
// ===== library: MasterCopy "Turbina" =====

FUNCTION_BLOCK "Turbina"   // FB1, LAD
{ S7_Optimized_Access := 'TRUE' }
VERSION : 0.1
   VAR_INPUT
      MotorAuxiliar : Bool;
      JuntaNeum : Bool;
      Frenos : Bool;
      Quemador_A : Bool;   // Entrada digital - Sensor Quemador A
      Quemador_B : Bool;   // Entrada digital - Sensor Quemador B
      Reset : Bool := False;
      ModoControl : Bool;   // Modo de control = 0=Manual 1=Auto
      SPManual : Int;   // Consigna manual
      SPAuto : Int;   // Consigna Automatica
   END_VAR
   VAR_OUTPUT
      SalidaVel : Int;
      SalidaPres : Int;
   END_VAR
   VAR_IN_OUT
      DB_Lazo : PID_Compact;
   END_VAR
   VAR
      Comando : Real;
      VelReal : Real;
      ValvReal : Real;
      ModeloPlanta : "ModeloPlanta";
      SP_ManualReal : Real;
      Valvula : Int;
      SP_AutoReal : Real;
   END_VAR
   VAR_TEMP
      KFrenos : Real;
      KMotor : Real;
      state : Int;
      error : Bool;
   END_VAR
   VAR_TEMP   // added for the SCL form of the ladder/FBD networks
      _w1 : Bool;
   END_VAR
BEGIN

REGION Network 1
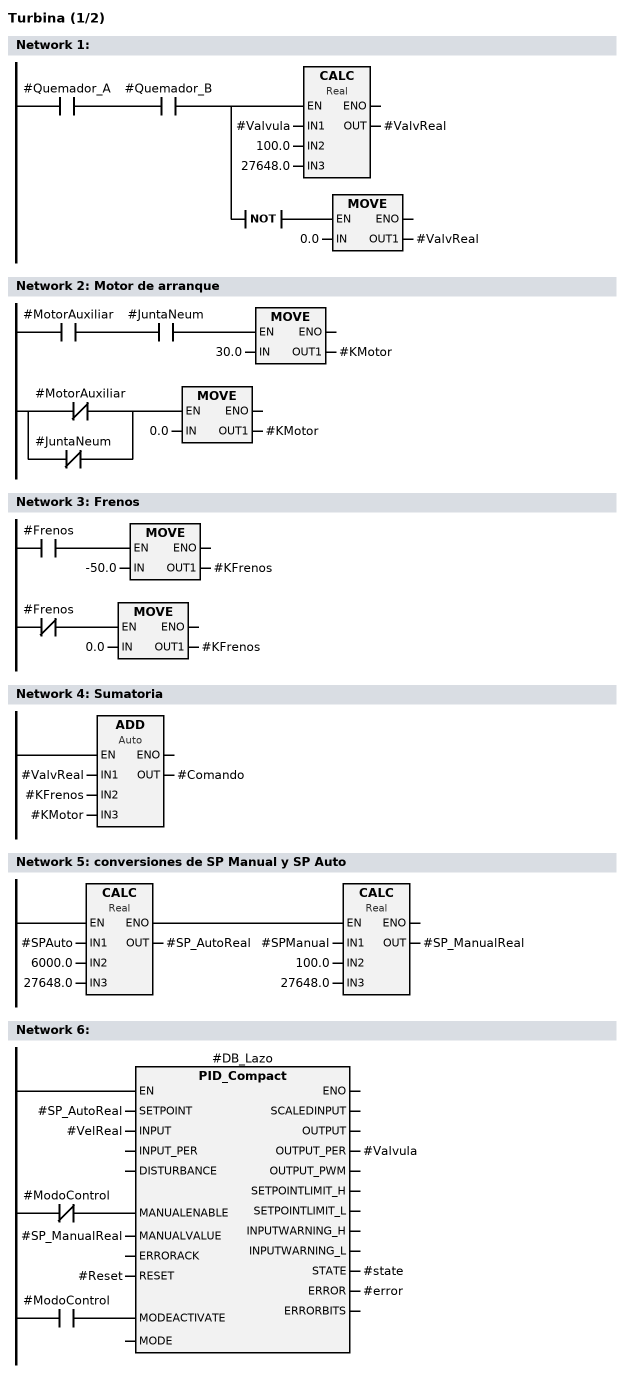
   #_w1 := #Quemador_A AND #Quemador_B;
   IF #_w1 THEN CALC(in1 := #Valvula, in2 := 100.0, in3 := 27648.0, out => #ValvReal); END_IF;
   IF NOT #_w1 THEN #ValvReal := 0.0; END_IF;
END_REGION

REGION Network 2: Motor de arranque
   RUNG wire#powerrail
      Contact( #MotorAuxiliar )
      Contact( #JuntaNeum )
      Move(in := 30.0, out1 => #KMotor)
   END_RUNG
   RUNG wire#powerrail
      I_Contact( #MotorAuxiliar )
      wire#w1
      Move(in := 0.0, out1 => #KMotor)
   END_RUNG
   RUNG wire#powerrail
      I_Contact( #JuntaNeum )
   END_RUNG wire#w1
   // the same network as SCL:
   IF #MotorAuxiliar AND #JuntaNeum THEN #KMotor := 30.0; END_IF;
   IF NOT #MotorAuxiliar OR NOT #JuntaNeum THEN #KMotor := 0.0; END_IF;
END_REGION

REGION Network 3: Frenos
   RUNG wire#powerrail
      Contact( #Frenos )
      Move(in := -50.0, out1 => #KFrenos)
   END_RUNG
   RUNG wire#powerrail
      I_Contact( #Frenos )
      Move(in := 0.0, out1 => #KFrenos)
   END_RUNG
   // the same network as SCL:
   IF #Frenos THEN #KFrenos := -50.0; END_IF;
   IF NOT #Frenos THEN #KFrenos := 0.0; END_IF;
END_REGION

REGION Network 4: Sumatoria
   RUNG wire#powerrail
      Add(in1 := #ValvReal, in2 := #KFrenos, in3 := #KMotor, out => #Comando)
   END_RUNG
   // the same network as SCL:
   #Comando := #ValvReal + #KFrenos + #KMotor;
END_REGION

REGION Network 5: conversiones de SP Manual y SP Auto
   CALC(in1 := #SPAuto, in2 := 6000.0, in3 := 27648.0, out => #SP_AutoReal);
   CALC(in1 := #SPManual, in2 := 100.0, in3 := 27648.0, out => #SP_ManualReal);
END_REGION

REGION Network 6
   #DB_Lazo(Setpoint := #SP_AutoReal,   // PID_Compact
            Input := #VelReal,
            ManualEnable := NOT #ModoControl,
            ManualValue := #SP_ManualReal,
            Reset := #Reset,
            ModeActivate := #ModoControl,
            Output_PER => #Valvula,
            State => #state,
            Error => #error);
END_REGION

REGION Network 7
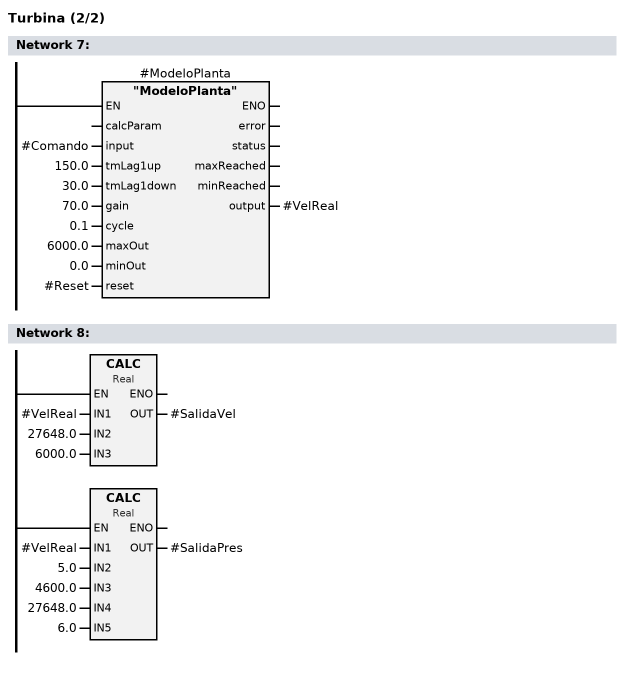
   RUNG wire#powerrail
      #ModeloPlanta(calcParam :=, input := #Comando, tmLag1up := 150.0, tmLag1down := 30.0, gain := 70.0, cycle := 0.1, maxOut := 6000.0, minOut := 0.0, reset := #Reset, error =>, status =>, maxReached =>, minReached =>, output => #VelReal)
   END_RUNG
   // the same network as SCL:
   #ModeloPlanta(input := #Comando,   // "ModeloPlanta"
                 tmLag1up := 150.0,
                 tmLag1down := 30.0,
                 gain := 70.0,
                 cycle := 0.1,
                 maxOut := 6000.0,
                 minOut := 0.0,
                 reset := #Reset,
                 output => #VelReal);
END_REGION

REGION Network 8
   CALC(in1 := #VelReal, in2 := 27648.0, in3 := 6000.0, out => #SalidaVel);
   CALC(in1 := #VelReal, in2 := 5.0, in3 := 4600.0, in4 := 27648.0, in5 := 6.0, out => #SalidaPres);
END_REGION
END_FUNCTION_BLOCK

// ===== library: MasterCopy "ModeloPlanta" =====

FUNCTION_BLOCK "ModeloPlanta"   // FB51, SCL
{ S7_Optimized_Access := 'TRUE' }
VERSION : 2.01
   VAR_INPUT
      calcParam : Bool;   // recalculate with new parameters
      input : Real;   // input signal
      tmLag1up : Real := 1.0;   // time constant T1 [sec] rising input
      tmLag1down : Real := 10.0;   // time constant T1 [sec] falling input
      gain : Real := 1.0;   // gain factor
      cycle : Real := 0.1;   // cyclic time [sec]
      maxOut : Real := 100.0;   // max. output limit
      minOut : Real;   // min. output limit
      reset : Bool;   // resets all relevant parameters to ‘0’ including the output
   END_VAR
   VAR_OUTPUT
      error : Bool;   // error (#tmLag1 <= 0 or #tmLag2 <= 0)
      status : Word;   // status (if #error = TRUE then status = 16#8001)
      maxReached : Bool;   // output has reached max. limit
      minReached : Bool;   // output has reached min. limit
      output : Real;   // output signal (if #error = FALSE)
   END_VAR
   VAR
      statRxn1 : Real;   // delayed input signal (n-1)
      statRyn1 : Real;   // delayed output signal (n-1)
      statRf1up : Real;   // Z-parameter 1 (rising xn)
      statRe1up : Real;   // Z-parameter 2 (rising xn)
      statRf1dn : Real;   // Z-parameter 1 (falling xn)
      statRe1dn : Real;   // Z-parameter 2 (falling xn)
      statRf1 : Real;   // active Z-parameter 1
      statRe1 : Real;   // active Z-parameter 2
      statOverfirst : Bool;
      statOutput : Real;
   END_VAR
BEGIN
   //=============================================================================
   //SIEMENS AG
   //(c)Copyright 2017 All Rights Reserved
   //-----------------------------------------------------------------------------
   //Library:       Library for Controlled System Simulation
   //Tested with:   S7-1500 FW V2.0 / S7-1200 FW V4.2
   //Engineering:   STEP 7 V14 Upd2 (TIA Portal)
   //Restrictions:  Cyclic interrupt
   //Requirements:  memory card needed for S7-1500
   //Functionality: Simulation of a PT1-System with two different Time-Constants
   //
   //  tmLag1up: Time-Constant for positive Inputsignal changes 
   //  tmLag1down: Time-Constant for negative Inputsignal changes
   //  
   //                gain
   //  Fup(p) = ----------------
   //           tmLag1up * p + 1
   //          
   //                    gain
   //  Fdown(p) = ------------------
   //             tmLag1down * p + 1
   //          
   //  Call the simulation in a cyclic interrupt with
   //  //  cyclic interrupt time at least = tmLag1/10!
   //-----------------------------------------------------------------------------
   //Change log table:
   //Version  Date       Expert in charge                Changes applied
   //02.00.00 03.02.2016 Siemens Industry Online Support Release (STEP 7 V13 SP1)
   //02.00.01 02.03.2017 Siemens Industry Online Support Release (STEP 7 V14)
   //=============================================================================

   // check parameter
   IF #tmLag1up <= 0 OR #tmLag1down <= 0 THEN
     #error := TRUE;
     #status := W#16#8001;     // Parameter Error
     #statOutput := 0;
     #output := 0;
     RETURN;
   ELSE
     #error := FALSE;
     #status := W#16#0000;     // no error
   END_IF;

   IF #calcParam = True OR NOT #statOverfirst THEN
     #statOverfirst:=1;
   // Z-parameters for Laplace PT1-System (rising signal change)
   #statRe1up := - EXP(-#cycle/#tmLag1up);
   #statRf1up := #gain*(1 + #statRe1up);
   // Z-parameters for Laplace PT1-System (falling signal change)
   #statRe1dn := - EXP(-#cycle/#tmLag1down);
   #statRf1dn := #gain*(1 + #statRe1dn);
   END_IF;

   // save delayed output signals
   #statRyn1:= #statOutput;

   // Change the parameter sets, dependent to Input Change
   IF (#input - #statRxn1) > 0 THEN
     #statRf1 := #statRf1up;
     #statRe1 := #statRe1up;
   ELSIF (#input - #statRxn1) < 0 THEN
      #statRf1 := #statRf1dn;
      #statRe1 := #statRe1dn;
   ELSE
     ;
   END_IF;

   // Differencial Equation of PT1-System
   #statOutput := #input*#statRf1 - #statRyn1*#statRe1;

   // save delayed input signals
   #statRxn1 := #input;

   // max limit of acutating variable
   IF #statOutput > #maxOut THEN
     #statOutput := #maxOut;
     #maxReached:= True;
   ELSE
     #maxReached := False;
   END_IF;

   // min limit of acutating variable
   IF #statOutput < #minOut THEN
     #statOutput := #minOut;
     #minReached := True;
   ELSE
     #minReached := False;
   END_IF;

   IF #reset THEN
     #statOutput := 0;
   END_IF;

   #output := #statOutput;
END_FUNCTION_BLOCK